// SIMATIC STEP 7 (V5.x) project Проба
// CPU: CPU 316-2 DP
// station: P_ADR_BUS
// station: Hardware
// station: SIMATIC 300(1)
// program: S7 Program(3)
// program: S7 Program(5)

FUNCTION FC 1 : VOID
TITLE = Счет готовых изделий
VERSION : 0.1
BEGIN
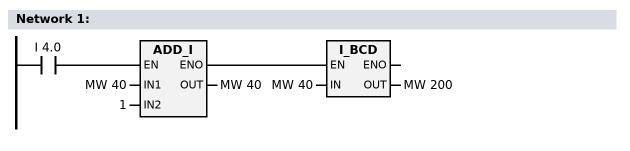
NETWORK
TITLE =
      A(;
      A     I 4.0;
      JNB   _001;
      L     MW 40;
      L     1;
      +I;
      T     MW 40;
      AN    OV;
      SAVE;
      CLR;
_001: A     BR;
      );
      JNB   _002;
      L     MW 40;
      ITB;
      T     MW 200;
_002: NOP   0;
END_FUNCTION

ORGANIZATION_BLOCK OB 1
TITLE = "Main Program Sweep (Cycle)"
VERSION : 0.1
VAR_TEMP
  OB1_EV_CLASS : BYTE ;	//Bits 0-3 = 1 (Coming event), Bits 4-7 = 1 (Event class 1)
  OB1_SCAN_1 : BYTE ;	//1 (Cold restart scan 1 of OB 1), 3 (Scan 2-n of OB 1)
  OB1_PRIORITY : BYTE ;	//Priority of OB Execution
  OB1_OB_NUMBR : BYTE ;	//1 (Organization block 1, OB1)
  OB1_RESERVED_1 : BYTE ;	//Reserved for system
  OB1_RESERVED_2 : BYTE ;	//Reserved for system
  OB1_PREV_CYCLE : INT ;	//Cycle time of previous OB1 scan (milliseconds)
  OB1_MIN_CYCLE : INT ;	//Minimum cycle time of OB1 (milliseconds)
  OB1_MAX_CYCLE : INT ;	//Maximum cycle time of OB1 (milliseconds)
  OB1_DATE_TIME : DATE_AND_TIME ;	//Date and time OB1 started
END_VAR
BEGIN
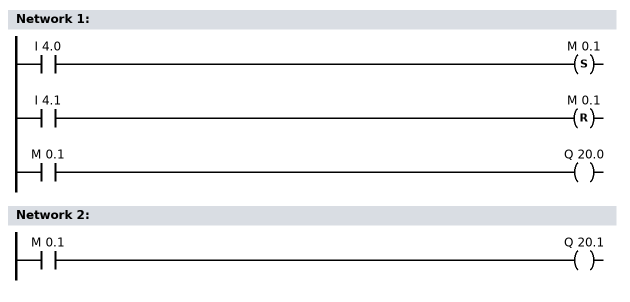
NETWORK
TITLE =
      A     I 4.0;
      S     M 0.1;
      A     I 4.1;
      R     M 0.1;
      A     M 0.1;
      =     Q 20.0;
NETWORK
TITLE =
      A     M 0.1;
      =     Q 20.1;
END_ORGANIZATION_BLOCK
